FUNCTION_BLOCK EL5102
VAR
	_io : EL5102_Data;
	{attribute addProperty Name "WcState"}
	_wcState : WcStateInputToggle;
	{attribute addProperty Name "Info data"}
	_infoData : InfoDataAdsDC;
END_VAR

PROPERTY IO : REFERENCE TO EL5102_Data
GET
IO REF= _io;
END_GET
END_PROPERTY

PROPERTY WcState : REFERENCE TO WcStateInputToggle
GET
WcState REF= _wcState;
END_GET
END_PROPERTY

END_FUNCTION_BLOCK

(* stored: Version 1.1.0.1, ProductVersion 3.1.4024.9
   POU EL5102: Id {c869de48-2e14-08ef-2fcc-ce5ebf2c4245}, SpecialFunc None
   Property IO: Id {bbcc8696-b157-0515-2fa9-ed11cf922f68}
   Get Get: Id {3b67e215-b5e6-01a8-39be-83a9d519d031}
   Property WcState: Id {c5eae1a7-9b15-053e-3229-2c12282c12e3}
   Get Get: Id {47aebfe7-83ed-0e07-3cf5-43d579b20c84} *)
